FUNCTION_BLOCK FB_CheckMessageBounds
VAR_IN_OUT
	iqArrayToCheck:typeMessage; //type of message bounds
	

END_VAR
VAR_OUTPUT
	qAnyMsgActive: BOOL;
	qMsgNumberActive: INT;
	
	qSingleMessage: STRING(255);
	
	qAllMessages: STRING;
	
	//special declare, follows typeMessageRowsArry
	qMsgRows:ARRAY[1..HMIData.gNumberOfMessagesScreen] OF typeMessageRow;
	

END_VAR
VAR
	i: INT;//for the loop
	lowestValue: UDINT :=4294967295; //set as init for highest possible value and work down from there
	lowestMessage: INT;
	allstrings: STRING;
	rollinglowestValue: UDINT :=0; //set as init for lowest possible value and work up
	newlineInsert: string;

	messageHeader: STRING(255);
	memcomparecheck: DINT;
	memchanged: BOOL;
	messagenum: DINT;
	strheader:STRING(255);
	
	n: UINT;
	returnclearing: UDINT;
	msgIndex: INT;
END_VAR

VAR_INPUT
	iMessageGroup: INT;
	isAlarm: BOOL; //for colour assigment
	isWarning: BOOL; //for colour assigment




END_VAR

	//mark active message as inactive
	//reset before scan
	actArraysMatch();
	

	
	
	
	
IF memchanged THEN //if the memory array have changed, then process the message
		
			//reset assumption that message is active
			qAnyMsgActive		:= FALSE;
			qMsgNumberActive 	:= 0;
			
			//clear down output alarm listing
			actCleanDownMsg();

	//may not need this
	FOR i := 0 TO GlobalMessages.gNumMessagesPerType DO
		
		//loop entire array
		IF iqArrayToCheck.message[i] = TRUE THEN
			//mark active message as active
			qAnyMsgActive		:= TRUE;
			qMsgNumberActive 	:= i;
		END_IF
			
		//move time of message into message type
		IF 			iqArrayToCheck.message[i] = TRUE 
			AND 	iqArrayToCheck.messageActive[i] = FALSE
			AND  iqArrayToCheck.messageTimeActive[i] = 0   
			THEN
				iqArrayToCheck.messageTimeActive[i] := System.myPlcInfoTask1.CycleCount;
			//write message text to array
		END_IF
		
		//find lowest message number, the lowest number is the first message that has appeared and thus, the only one worthwhile
		IF qAnyMsgActive THEN //if there is any message active in the array, then find the lowest number
			IF iqArrayToCheck.messageTimeActive[i] > 1 THEN 			//consider the message
				IF  iqArrayToCheck.messageTimeActive[i] < lowestValue   THEN
					//record the index of the lowest message to write later
					lowestValue := 	iqArrayToCheck.messageTimeActive[i];//lowest TIME value
					lowestMessage := i;									//lowest value message		
					qSingleMessage := iqArrayToCheck.text[i];			//return the message text of the single lowest alarm
					
					IF rollinglowestValue = 0 THEN //starting point
						rollinglowestValue := lowestValue;				//assign lowest message for multi line use
					END_IF
				
				END_IF	
			END_IF
		ELSE
			//no message active at all, so return zeros
			qSingleMessage := 'no message';								//no message text
			lowestMessage := 0;											//return zero for no message
			lowestValue := 4294967295;									//return highest possible number for next time
			
			//clear down single data
			qAnyMsgActive		:= FALSE;								//clear down with implicit
			qMsgNumberActive 	:= 0;									//clear down with implicit
			rollinglowestValue 	:= 0;
		END_IF
		/////////////////////////////////////////////////////////////////////////////////////////////////////////////////////////////
		//loop around the array and find the lowest number >1 and write that message first, then all other messages in incrementing order
		//once the message is written to the list, set the .MessageActive bit to TRUE
		IF rollinglowestValue > 1 THEN //rolling value is valid
			
			//the current message is active, but not yet written
			IF iqArrayToCheck.message[i] = TRUE  THEN
				
								//combine message texts into long string with CR LFs
								newlineInsert := concat(iqArrayToCheck.text[i], '$0D'); //make new line
								
								//calc message number
								messagenum := iMessageGroup + i; //creates 10000 + 1, 10001 mesage number
								
								//string header
								strheader := concat(DINT_TO_STRING(messagenum), ' '); //'10001 ' with space
								
								//add message number
								newlineInsert := concat(strheader,newlineInsert);
									 
								allstrings := concat(newlineInsert,allstrings); //and put it at the top of the pack
								
								//message was written, so turn on message active bit iqArrayToCheck.messageActive[i]
								iqArrayToCheck.messageActive[i] := TRUE;
								
								
						
			END_IF	
			
		END_IF
		
		//reset message usage on dual arrays
		IF iqArrayToCheck.message[i] = FALSE AND  iqArrayToCheck.messageActive[i] = TRUE THEN
		iqArrayToCheck.messageActive[i] := FALSE;
		iqArrayToCheck.messageTimeActive[i] := 0;
		END_IF
		
		//message exists, so write strings to output
		IF rollinglowestValue > 1 THEN 
					qAllMessages := allstrings;
				ELSE
					newlineInsert := '';
					allstrings := '';
					qAllMessages:= '';
		END_IF
		
	
	END_FOR;

	//fill alarm rows
//	FOR n := 0 TO HMIData.gNumberOfMessagesScreen DO
	//	qMsgRows.AlarmViewMsg[n].msgText := '';
			
//	END_FOR
END_IF


msgindex := 1;
IF memchanged THEN
	FOR i := 0 TO GlobalMessages.gNumMessagesPerType DO
		
			//find next TRUE alarm
			IF iqArrayToCheck.messageActive[i] = TRUE THEN
				
				//assign text to other alarm view 	
				qMsgRows[msgindex].msgText := iqArrayToCheck.text[i];
				
				//assign colour
				IF isAlarm THEN
					qMsgRows[msgIndex].isAlarm := TRUE;
					ELSE
					qMsgRows[msgIndex].isAlarm := FALSE;	
				
				END_IF
				
					//assign colour
				IF isWarning THEN
					qMsgRows[msgIndex].isWarning := TRUE;
					ELSE
					qMsgRows[msgIndex].isWarning := FALSE;
				
				END_IF
				
				//increment message index and try again
				msgindex := msgIndex + 1;
			
				//exit loop 
				IF msgIndex > GlobalMessages.gNumMessagesPerType - 1 THEN
					EXIT;
				END_IF
				
			END_IF
		
	END_FOR


END_IF

ACTION actArraysMatch:
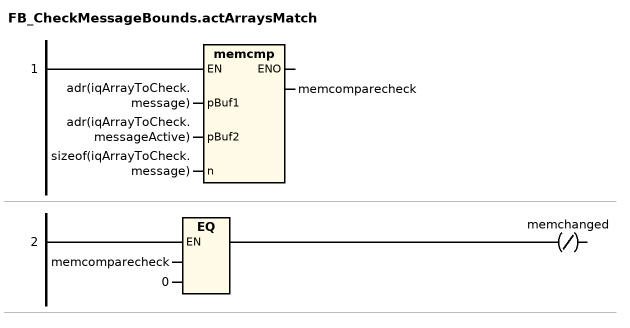
// NETWORK 1
memcomparecheck := memcmp(pBuf1 := adr(iqArrayToCheck.message), pBuf2 := adr(iqArrayToCheck.messageActive), n := sizeof(iqArrayToCheck.message));

// NETWORK 2
memchanged := NOT (memcomparecheck = 0);
END_ACTION

ACTION actCleanDownMsg:
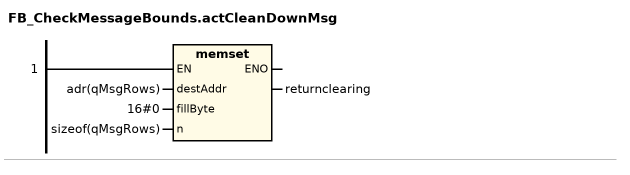
// NETWORK 1
returnclearing := memset(destAddr := adr(qMsgRows), fillByte := 16#0, n := sizeof(qMsgRows));
END_ACTION

END_FUNCTION_BLOCK

(* stored: Version 1.1.0.1, ProductVersion 3.1.4024.12
   POU FB_CheckMessageBounds: Id {cfd3e64b-34a3-43a4-b491-e0f565bbe474}, SpecialFunc None
   Action actArraysMatch: Id {deaf4cea-369a-4b23-adf0-691b3612839c}
   Action actCleanDownMsg: Id {c459896b-96a2-4e11-8e93-84fa94812ca5} *)
